// TIA Portal V19 export
TYPE "Positioning_DOL_Machine_Par"
// stored: Access Published
   STRUCT
      PosTolerance { S7_SetPoint := 'True'} : LReal;   // mm
      Minus_Limit { S7_SetPoint := 'True'} : LReal;   // mm
      Plus_Limit { S7_SetPoint := 'True'} : LReal;   // mm
      PreCutOff { S7_SetPoint := 'True'} : LReal;   // mm
      PreEndLowSpeed { S7_SetPoint := 'True'} : LReal;   // mm
      PreEndMedSpeed { S7_SetPoint := 'True'} : LReal;   // mm
      LowSpeed { S7_SetPoint := 'True'} : LReal;   // % di speed massima
      MedSpeed { S7_SetPoint := 'True'} : LReal;   // % di speed massima
      HighSpeed { S7_SetPoint := 'True'} : LReal;   // % di speed massima
      Man_Speed { S7_SetPoint := 'True'} : LReal;   // Velocità manuale [1-100%]
   END_STRUCT;
END_TYPE
